(* IEC 61131-3 sources: Controller/, 6 files *)

(* ----  Codesys.ST ---- *)
(* ============================================
   КЕРУВАННЯ БОЙЛЕРОМ / ГАЗОВИМ ОБЛАДНАННЯМ
   Codesys 3.5 — Structured Text (ST)

   Як створити проект в Codesys:
   1. File → New Project → Standard Project
   2. Вибрати свій контролер або "CODESYS Control Win" для симуляції
   3. У дереві проекту: двічі клікнути PLC_PRG
   4. Вставити цей код
   5. Build → Build Solution (F11)
   6. Online → Login (Alt+F8) → Start (F5)
   ============================================ *)

PROGRAM PLC_PRG
VAR
    (* ==========================================
       АНАЛОГОВІ ВХОДИ (підключаються через
       Codesys I/O Mapping до реальних каналів)
       ========================================== *)
    AI_NAPRUGA      : INT;   (* Напруга бойлера, АЦП 0-4095 = 0-500В *)
    AI_TEMP_BOILER  : INT;   (* Температура бойлера, АЦП 0-4095 = 0-150°C *)
    AI_TEMP_VODA    : INT;   (* Температура води, АЦП 0-4095 = 0-150°C *)
    AI_TEMP_2       : INT;   (* Додатковий датчик температури *)
    AI_TISK_MASLA   : INT;   (* Тиск масла аналоговий, АЦП 0-4095 *)

    (* ==========================================
       ДИСКРЕТНІ ВХОДИ
       ========================================== *)
    X_GAZ           : BOOL;  (* Датчик газу: TRUE=є газ (замкнутий) *)
    X_VAKUUM        : BOOL;  (* Датчик вакууму: TRUE=є вакуум (замкнутий) *)
    X_TISK_MASLA_DI : BOOL;  (* Тиск масла: TRUE=норма (замкнутий) *)
    X_AVARIA_EXT    : BOOL;  (* Зовнішній аварійний СТОП *)

    (* ==========================================
       ДИСКРЕТНІ ВИХОДИ
       ========================================== *)
    Y_KLAPAN_GAZ    : BOOL;  (* Клапан газу: TRUE=відкрито *)
    Y_ROZET_1       : BOOL;  (* Розетка 1 *)
    Y_ROZET_2       : BOOL;  (* Розетка 2 *)
    Y_AVARIA_SIGNAL : BOOL;  (* Аварійна сигналізація (лампа/сирена) *)
    Y_DOZV_ROBOTY   : BOOL;  (* Загальний дозвіл роботи *)

    (* ==========================================
       КОМАНДИ ОПЕРАТОРА (з HMI або Visualization)
       ========================================== *)
    CMD_START       : BOOL;  (* Кнопка СТАРТ *)
    CMD_STOP        : BOOL;  (* Кнопка СТОП *)
    CMD_ROZET_1     : BOOL;  (* Команда увімкнути розетку 1 *)
    CMD_ROZET_2     : BOOL;  (* Команда увімкнути розетку 2 *)
    CMD_RESET_AVAR  : BOOL;  (* Скидання аварії вручну *)

    (* ==========================================
       ВНУТРІШНІ ЗМІННІ — АВАРІЇ
       ========================================== *)
    M_AVARIA_NAPRUGA    : BOOL;  (* Аварія: напруга >= 400В *)
    M_AVARIA_TEMP       : BOOL;  (* Аварія: температура бойлера >= 80°C *)
    M_AVARIA_VAKUUM     : BOOL;  (* Аварія: пропав вакуум *)
    M_ZAGALNA_AVARIA    : BOOL;  (* Загальна аварія (будь-яка з вище) *)

    (* ==========================================
       ВНУТРІШНІ ЗМІННІ — СТАНИ ДАТЧИКІВ
       ========================================== *)
    M_GAZ_IE            : BOOL;  (* Газ є = TRUE, немає = FALSE *)
    M_VAKUUM_IE         : BOOL;  (* Вакуум є = TRUE, немає = FALSE *)
    M_TISK_NORMA        : BOOL;  (* Тиск масла норма = TRUE *)

    (* ==========================================
       ВНУТРІШНІ ЗМІННІ — СИСТЕМА
       ========================================== *)
    M_SYSTEM_ON         : BOOL;  (* Система запущена оператором *)
    M_SYSTEM_READY      : BOOL;  (* Система готова до роботи *)

    (* ==========================================
       РЕАЛЬНІ ЗНАЧЕННЯ ДЛЯ ВІДОБРАЖЕННЯ НА HMI
       ========================================== *)
    NAPRUGA_VOLT        : INT;   (* Напруга в Вольтах *)
    TEMP_BOILER_GRAD    : INT;   (* Температура бойлера в °C *)
    TEMP_VODA_GRAD      : INT;   (* Температура води в °C *)
    TEMP_2_GRAD         : INT;   (* Температура доп. датчика в °C *)

    (* ==========================================
       ДОПОМІЖНІ ТРИГЕРИ (для кнопок START/STOP)
       ========================================== *)
    trig_START          : R_TRIG;  (* Фронт сигналу СТАРТ *)
    trig_STOP           : R_TRIG;  (* Фронт сигналу СТОП *)
    trig_RESET          : R_TRIG;  (* Фронт сигналу СКИДАННЯ *)
END_VAR

(* ============================================================
   БЛОК 1: ОБРОБКА КНОПОК СТАРТ / СТОП
   R_TRIG реагує тільки на момент натискання (фронт сигналу)
   ============================================================ *)
trig_START(CLK := CMD_START);
trig_STOP(CLK  := CMD_STOP);
trig_RESET(CLK := CMD_RESET_AVAR);

(* Запуск системи — тільки якщо немає аварії *)
IF trig_START.Q AND NOT M_ZAGALNA_AVARIA THEN
    M_SYSTEM_ON := TRUE;
END_IF;

(* Зупинка системи *)
IF trig_STOP.Q OR M_ZAGALNA_AVARIA THEN
    M_SYSTEM_ON := FALSE;
END_IF;

(* ============================================================
   БЛОК 2: ПЕРЕРАХУНОК АЦП → РЕАЛЬНІ ОДИНИЦІ

   Формула: РЕАЛЬНЕ = АЦП_ЗНАЧЕННЯ * МАКСИМУМ / 4095

   АЦП дає число від 0 до 4095 (12-бітний)
   Це число відповідає реальному вхідному сигналу 0-10В або 4-20мА
   ============================================================ *)

(* Напруга бойлера: вхід 0-10В = 0-500В реальних *)
NAPRUGA_VOLT     := INT_TO_INT(REAL_TO_INT(INT_TO_REAL(AI_NAPRUGA) * 500.0 / 4095.0));

(* Температура бойлера: вхід 4-20мА через модуль = 0-150°C *)
TEMP_BOILER_GRAD := INT_TO_INT(REAL_TO_INT(INT_TO_REAL(AI_TEMP_BOILER) * 150.0 / 4095.0));

(* Температура води *)
TEMP_VODA_GRAD   := INT_TO_INT(REAL_TO_INT(INT_TO_REAL(AI_TEMP_VODA) * 150.0 / 4095.0));

(* Додатковий датчик температури *)
TEMP_2_GRAD      := INT_TO_INT(REAL_TO_INT(INT_TO_REAL(AI_TEMP_2) * 150.0 / 4095.0));

(* ============================================================
   БЛОК 3: АВАРІЯ ПО НАПРУЗІ БОЙЛЕРА

   УМОВА: якщо напруга >= 400В → АВАРІЯ → все зупиняється
   ГІСТЕРЕЗИС: скидається тільки якщо впала нижче 380В
   (щоб уникнути постійного вмикання/вимикання на межі 400В)
   ============================================================ *)
IF NAPRUGA_VOLT >= 400 THEN
    M_AVARIA_NAPRUGA := TRUE;
ELSIF NAPRUGA_VOLT < 380 THEN
    (* Скидати аварію автоматично тільки якщо напруга впала *)
    (* Якщо хочеш скидати тільки вручну — закоментуй цей рядок *)
    IF trig_RESET.Q THEN
        M_AVARIA_NAPRUGA := FALSE;
    END_IF;
END_IF;

(* ============================================================
   БЛОК 4: АВАРІЯ ПО ТЕМПЕРАТУРІ БОЙЛЕРА

   УМОВА: якщо температура >= 80°C → АВАРІЯ → все зупиняється
   ГІСТЕРЕЗИС: скидається тільки якщо охолонув нижче 75°C
   ============================================================ *)
IF TEMP_BOILER_GRAD >= 80 THEN
    M_AVARIA_TEMP := TRUE;
ELSIF TEMP_BOILER_GRAD < 75 THEN
    IF trig_RESET.Q THEN
        M_AVARIA_TEMP := FALSE;
    END_IF;
END_IF;

(* ============================================================
   БЛОК 5: ДАТЧИК ГАЗУ

   X_GAZ = TRUE  (замкнутий контакт) → газ є   → M_GAZ_IE = 1
   X_GAZ = FALSE (розімкнутий)       → газу немає → M_GAZ_IE = 0

   На HMI відображати: якщо M_GAZ_IE=TRUE показуй "1 - ГАЗ Є"
                        якщо M_GAZ_IE=FALSE показуй "0 - ГАЗУ НЕМАЄ"
   ============================================================ *)
M_GAZ_IE := X_GAZ;

(* ============================================================
   БЛОК 6: ДАТЧИК ВАКУУМУ

   X_VAKUUM = TRUE  (замкнутий) → вакуум є   → робота дозволена
   X_VAKUUM = FALSE (розімкнутий) → вакууму немає → ЗУПИНКА + ЗАКРИТИ ГАЗ
   ============================================================ *)
M_VAKUUM_IE := X_VAKUUM;

IF NOT M_VAKUUM_IE THEN
    M_AVARIA_VAKUUM := TRUE;   (* Немає вакууму — АВАРІЯ *)
ELSE
    M_AVARIA_VAKUUM := FALSE;  (* Вакуум є — норма *)
END_IF;

(* ============================================================
   БЛОК 7: ДАТЧИК ТИСКУ МАСЛА

   X_TISK_MASLA_DI = TRUE  (замкнутий) → тиск норма
   X_TISK_MASLA_DI = FALSE (розімкнутий) → тиск низький → АВАРІЯ
   ============================================================ *)
M_TISK_NORMA := X_TISK_MASLA_DI;

(* ============================================================
   БЛОК 8: ЗАГАЛЬНА АВАРІЯ

   Якщо БУДЬ-ЯКА з умов виконана → загальна аварія
   → система зупиняється
   → клапан газу закривається
   → вмикається сигналізація
   ============================================================ *)
M_ZAGALNA_AVARIA := M_AVARIA_NAPRUGA    (* Напруга >= 400В *)
                 OR M_AVARIA_TEMP        (* Температура >= 80°C *)
                 OR M_AVARIA_VAKUUM      (* Немає вакууму *)
                 OR NOT M_TISK_NORMA     (* Тиск масла низький *)
                 OR X_AVARIA_EXT;        (* Зовнішній аварійний стоп *)

(* ============================================================
   БЛОК 9: ГОТОВНІСТЬ СИСТЕМИ ДО РОБОТИ

   ВСІ умови мають бути виконані одночасно:
   ✓ Напруга норма (< 400В)
   ✓ Температура норма (< 80°C)
   ✓ Газ є
   ✓ Вакуум є  ← НАЙВАЖЛИВІШЕ
   ✓ Тиск масла норма
   ✓ Немає зовнішньої аварії
   ✓ Оператор натиснув СТАРТ
   ============================================================ *)
M_SYSTEM_READY := NOT M_AVARIA_NAPRUGA
              AND NOT M_AVARIA_TEMP
              AND M_GAZ_IE
              AND M_VAKUUM_IE
              AND M_TISK_NORMA
              AND NOT X_AVARIA_EXT
              AND M_SYSTEM_ON;

(* ============================================================
   БЛОК 10: КЕРУВАННЯ КЛАПАНОМ ГАЗУ

   ВІДКРИТИ газ → тільки якщо система готова (всі умови ОК)
   ЗАКРИТИ газ → при будь-якій аварії, і особливо при відсутності вакууму

   БЕЗПЕКА: подвійна перевірка вакууму — навіть якщо
   щось пішло не так в логіці вище, газ все одно закриється
   ============================================================ *)
IF M_SYSTEM_READY THEN
    Y_KLAPAN_GAZ := TRUE;    (* Відкрити клапан газу *)
ELSE
    Y_KLAPAN_GAZ := FALSE;   (* Закрити клапан газу *)
END_IF;

(* КРИТИЧНА БЕЗПЕКА: подвійна гарантія закриття газу без вакууму *)
IF NOT M_VAKUUM_IE THEN
    Y_KLAPAN_GAZ := FALSE;   (* ОБОВ'ЯЗКОВО закрити! *)
END_IF;

(* КРИТИЧНА БЕЗПЕКА: закрити газ при аварії напруги або температури *)
IF M_AVARIA_NAPRUGA OR M_AVARIA_TEMP THEN
    Y_KLAPAN_GAZ := FALSE;
END_IF;

(* ============================================================
   БЛОК 11: КЕРУВАННЯ РОЗЕТКАМИ

   Розетки вмикаються командою оператора (з HMI або кнопки)
   АЛЕ тільки якщо немає загальної аварії
   ============================================================ *)
IF CMD_ROZET_1 AND NOT M_ZAGALNA_AVARIA THEN
    Y_ROZET_1 := TRUE;
ELSE
    Y_ROZET_1 := FALSE;
END_IF;

IF CMD_ROZET_2 AND NOT M_ZAGALNA_AVARIA THEN
    Y_ROZET_2 := TRUE;
ELSE
    Y_ROZET_2 := FALSE;
END_IF;

(* ============================================================
   БЛОК 12: АВАРІЙНА СИГНАЛІЗАЦІЯ
   Лампа або сирена вмикається при будь-якій аварії
   ============================================================ *)
Y_AVARIA_SIGNAL := M_ZAGALNA_AVARIA;

(* ============================================================
   БЛОК 13: ЗАГАЛЬНИЙ ДОЗВІЛ РОБОТИ
   Цей вихід можна підключити до загального контактора
   ============================================================ *)
Y_DOZV_ROBOTY := M_SYSTEM_READY;

END_PROGRAM

(* ---- BoilerController.ST ---- *)
(* ============================================
   КОНТРОЛЕР УПРАВЛІННЯ БОЙЛЕРОМ
   FATEK FBs-MA - Structured Text (ST)
   Версія 2.0 - Оптимізований під ваші вимоги
   ============================================ *)

(* --- КОНСТАНТИ --- *)
VAR CONSTANT
    (* Діапазони АЦП *)
    ADC_MAX         : INT := 4095;
    VOLTAGE_MAX     : INT := 500;   (* Макс. напруга, В *)
    TEMP_MAX        : INT := 150;   (* Макс. температура, °C *)

    (* Аварійні межі *)
    VOLTAGE_ALARM   : INT := 400;   (* Аварія напруги при 400В *)
    VOLTAGE_RESET   : INT := 380;   (* Скидання при 380В *)
    TEMP_ALARM      : INT := 80;    (* Аварія температури при 80°C *)
    TEMP_RESET      : INT := 75;    (* Скидання при 75°C *)

    (* АЦП значення для аварій *)
    ADC_VOLTAGE_ALARM : INT := 3276; (* 400В → АЦП: 4095*400/500 *)
    ADC_TEMP_ALARM    : INT := 2184; (* 80°C → АЦП: 4095*80/150 *)
END_VAR

(* --- ВХОДИ (Inputs) --- *)
VAR
    (* Аналогові входи 0..4095 *)
    AI_VOLTAGE      AT %IW0 : INT;   (* Напруга бойлера 0-500В *)
    AI_TEMP_BOILER  AT %IW1 : INT;   (* Температура бойлера 0-150°C *)
    AI_TEMP_WATER   AT %IW2 : INT;   (* Температура води 0-150°C *)
    AI_TEMP_1       AT %IW3 : INT;   (* Датчик температури 1 *)
    AI_TEMP_2       AT %IW4 : INT;   (* Датчик температури 2 *)
    AI_OIL_PRESSURE AT %IW5 : INT;   (* Тиск масла (аналоговий) *)

    (* Дискретні входи *)
    X_GAS_PRESENT   AT %IX0.0 : BOOL; (* Датчик газу: TRUE=є газ *)
    X_VACUUM_OK     AT %IX0.1 : BOOL; (* Датчик вакууму: TRUE=є вакуум *)
    X_OIL_PRESS_OK  AT %IX0.2 : BOOL; (* Тиск масла: TRUE=норма *)
    X_EMERGENCY_STOP: AT %IX0.3 : BOOL; (* Аварійний стоп: TRUE=активний *)

    (* Команди оператора/HMI *)
    CMD_START       AT %MX10.0 : BOOL; (* Команда старт *)
    CMD_STOP        AT %MX10.1 : BOOL; (* Команда стоп *)
    CMD_SOCKET1     AT %MX10.2 : BOOL; (* Команда розетка 1 *)
    CMD_SOCKET2     AT %MX10.3 : BOOL; (* Команда розетка 2 *)
END_VAR

(* --- ВИХОДИ (Outputs) --- *)
VAR
    Y_GAS_VALVE     AT %QX0.0 : BOOL; (* Клапан газу: TRUE=відкрито *)
    Y_SOCKET1       AT %QX0.1 : BOOL; (* Розетка 1 *)
    Y_SOCKET2       AT %QX0.2 : BOOL; (* Розетка 2 *)
    Y_ALARM_LIGHT   AT %QX0.3 : BOOL; (* Аварійна лампа *)
    Y_PERMIT_RUN    AT %QX0.4 : BOOL; (* Дозвіл роботи *)
    Y_WATER_PUMP    AT %QX0.5 : BOOL; (* Насос води *)
END_VAR

(* --- ВНУТРІШНІ МАРКЕРИ --- *)
VAR
    (* Аварійні флаги *)
    M_VOLTAGE_ALARM : BOOL := FALSE; (* Аварія напруги *)
    M_TEMP_ALARM    : BOOL := FALSE; (* Аварія температури *)
    M_VACUUM_ALARM  : BOOL := FALSE; (* Аварія вакууму *)
    M_OIL_ALARM     : BOOL := FALSE; (* Аварія тиску масла *)
    M_ANY_ALARM     : BOOL := FALSE; (* Будь-яка аварія *)

    (* Стан системи *)
    M_SYSTEM_RUN    : BOOL := FALSE; (* Система запущена *)
    M_SYSTEM_READY  : BOOL := FALSE; (* Система готова *)
    M_GAS_AVAILABLE : BOOL := FALSE; (* Газ доступний *)
    M_VACUUM_OK     : BOOL := FALSE; (* Вакуум в нормі *)

    (* Фізичні величини для HMI *)
    VOLTAGE_DISPLAY : INT; (* Напруга в Вольтах *)
    TEMP_B_DISPLAY  : INT; (* Температура бойлера °C *)
    TEMP_W_DISPLAY  : INT; (* Температура води °C *)
    TEMP_1_DISPLAY  : INT; (* Температура датчик 1 °C *)
    TEMP_2_DISPLAY  : INT; (* Температура датчик 2 °C *)
    OIL_P_DISPLAY   : INT; (* Тиск масла в ум.од.*)

    (* Детектори фронтів *)
    M_CMD_START_OLD : BOOL := FALSE;
    M_CMD_STOP_OLD  : BOOL := FALSE;
    M_GAS_OLD       : BOOL := FALSE;
    M_VAC_OLD       : BOOL := FALSE;
    M_ALARM_OLD     : BOOL := FALSE;

    (* Статистика для HMI *)
    STAT_START_COUNT: INT := 0;
    STAT_ALARM_COUNT: INT := 0;
    STAT_GAS_OFF    : INT := 0;
    STAT_VAC_OFF    : INT := 0;
END_VAR

(* ============================================
   БЛОК 1: ПЕРЕТВОРЕННЯ АЦП → ФІЗИЧНІ ВЕЛИЧИНИ
   ============================================ *)

(* Напруга: 0-4095 = 0-500В *)
VOLTAGE_DISPLAY := AI_VOLTAGE * VOLTAGE_MAX / ADC_MAX;

(* Температури: 0-4095 = 0-150°C *)
TEMP_B_DISPLAY := AI_TEMP_BOILER * TEMP_MAX / ADC_MAX;
TEMP_W_DISPLAY := AI_TEMP_WATER * TEMP_MAX / ADC_MAX;
TEMP_1_DISPLAY := AI_TEMP_1 * TEMP_MAX / ADC_MAX;
TEMP_2_DISPLAY := AI_TEMP_2 * TEMP_MAX / ADC_MAX;

(* Тиск масла: 0-4095 = 0-100% *)
OIL_P_DISPLAY := AI_OIL_PRESSURE * 100 / ADC_MAX;

(* ============================================
   БЛОК 2: АВАРІЯ НАПРУГИ (≥400В)
   ============================================ *)
IF VOLTAGE_DISPLAY >= VOLTAGE_ALARM THEN
    M_VOLTAGE_ALARM := TRUE;
ELSE
    IF VOLTAGE_DISPLAY < VOLTAGE_RESET THEN
        M_VOLTAGE_ALARM := FALSE;
    END_IF;
END_IF;

(* ============================================
   БЛОК 3: АВАРІЯ ТЕМПЕРАТУРИ (≥80°C)
   ============================================ *)
IF TEMP_B_DISPLAY >= TEMP_ALARM THEN
    M_TEMP_ALARM := TRUE;
ELSE
    IF TEMP_B_DISPLAY < TEMP_RESET THEN
        M_TEMP_ALARM := FALSE;
    END_IF;
END_IF;

(* ============================================
   БЛОК 4: ДАТЧИК ГАЗУ
   ============================================ *)
M_GAS_AVAILABLE := X_GAS_PRESENT;

(* Лічильник відключень газу *)
IF M_GAS_AVAILABLE = FALSE AND M_GAS_OLD = TRUE THEN
    STAT_GAS_OFF := STAT_GAS_OFF + 1;
END_IF;
M_GAS_OLD := M_GAS_AVAILABLE;

(* ============================================
   БЛОК 5: ДАТЧИК ВАКУУМУ
   ============================================ *)
M_VACUUM_OK := X_VACUUM_OK;

IF M_VACUUM_OK = FALSE THEN
    M_VACUUM_ALARM := TRUE;  (* Немає вакууму = аварія *)
ELSE
    M_VACUUM_ALARM := FALSE;
END_IF;

(* Лічильник відключень вакууму *)
IF M_VACUUM_OK = FALSE AND M_VAC_OLD = TRUE THEN
    STAT_VAC_OFF := STAT_VAC_OFF + 1;
END_IF;
M_VAC_OLD := M_VACUUM_OK;

(* ============================================
   БЛОК 6: ТИСК МАСЛА
   ============================================ *)
IF X_OIL_PRESS_OK = FALSE THEN
    M_OIL_ALARM := TRUE;
ELSE
    M_OIL_ALARM := FALSE;
END_IF;

(* ============================================
   БЛОК 7: ЗАГАЛЬНА АВАРІЯ
   ============================================ *)
M_ANY_ALARM := M_VOLTAGE_ALARM
             OR M_TEMP_ALARM
             OR M_VACUUM_ALARM
             OR M_OIL_ALARM
             OR X_EMERGENCY_STOP;

(* Лічильник аварій *)
IF M_ANY_ALARM = TRUE AND M_ALARM_OLD = FALSE THEN
    STAT_ALARM_COUNT := STAT_ALARM_COUNT + 1;
END_IF;
M_ALARM_OLD := M_ANY_ALARM;

(* ============================================
   БЛОК 8: ЛОГІКА СТАРТ/СТОП
   ============================================ *)

(* Детектор фронту старту *)
IF CMD_START = TRUE AND M_CMD_START_OLD = FALSE THEN
    IF M_SYSTEM_RUN = FALSE AND M_ANY_ALARM = FALSE THEN
        M_SYSTEM_RUN := TRUE;
        STAT_START_COUNT := STAT_START_COUNT + 1;
    END_IF;
END_IF;
M_CMD_START_OLD := CMD_START;

(* Детектор фронту стопу *)
IF CMD_STOP = TRUE AND M_CMD_STOP_OLD = FALSE THEN
    M_SYSTEM_RUN := FALSE;
END_IF;
M_CMD_STOP_OLD := CMD_STOP;

(* Автоматичний стоп при аварії *)
IF M_ANY_ALARM = TRUE THEN
    M_SYSTEM_RUN := FALSE;
END_IF;

(* ============================================
   БЛОК 9: ГОТОВНІСТЬ СИСТЕМИ
   ============================================ *)
M_SYSTEM_READY := NOT M_VOLTAGE_ALARM      (* Напруга норма *)
                AND NOT M_TEMP_ALARM        (* Температура норма *)
                AND M_GAS_AVAILABLE          (* Газ є *)
                AND M_VACUUM_OK              (* Вакуум є *)
                AND NOT M_OIL_ALARM           (* Тиск масла норма *)
                AND NOT X_EMERGENCY_STOP      (* Немає аварійного стопу *)
                AND M_SYSTEM_RUN;             (* Система запущена *)

(* ============================================
   БЛОК 10: КЕРУВАННЯ КЛАПАНОМ ГАЗУ
   ============================================ *)
(* Головна логіка: газ відкритий тільки якщо ВСІ умови виконані *)
IF M_SYSTEM_READY THEN
    Y_GAS_VALVE := TRUE;   (* Відкрити клапан газу *)
ELSE
    Y_GAS_VALVE := FALSE;  (* Закрити клапан газу *)
END_IF;

(* Додатковий захист: якщо немає вакууму - ОБОВ'ЯЗКОВО закрити газ *)
IF M_VACUUM_OK = FALSE THEN
    Y_GAS_VALVE := FALSE;
END_IF;

(* ============================================
   БЛОК 11: КЕРУВАННЯ РОЗЕТКАМИ
   ============================================ *)

(* Розетка 1 - вмикається командою, але не при аварії *)
IF CMD_SOCKET1 = TRUE AND M_ANY_ALARM = FALSE THEN
    Y_SOCKET1 := TRUE;
ELSE
    Y_SOCKET1 := FALSE;
END_IF;

(* Розетка 2 - вмикається командою, але не при аварії *)
IF CMD_SOCKET2 = TRUE AND M_ANY_ALARM = FALSE THEN
    Y_SOCKET2 := TRUE;
ELSE
    Y_SOCKET2 := FALSE;
END_IF;

(* ============================================
   БЛОК 12: КЕРУВАННЯ НАСОСОМ ВОДИ
   ============================================ *)
(* Насос води працює якщо система готова і є температура води *)
IF M_SYSTEM_READY AND TEMP_W_DISPLAY > 20 THEN
    Y_WATER_PUMP := TRUE;
ELSE
    Y_WATER_PUMP := FALSE;
END_IF;

(* ============================================
   БЛОК 13: АВАРІЙНА СИГНАЛІЗАЦІЯ
   ============================================ *)
Y_ALARM_LIGHT := M_ANY_ALARM;

(* ============================================
   БЛОК 14: ЗАГАЛЬНИЙ ДОЗВІЛ РОБОТИ
   ============================================ *)
Y_PERMIT_RUN := M_SYSTEM_READY;

(* ============================================
   БЛОК 15: ЕКСПОРТ ДАНИХ ДЛЯ HMI
   ============================================ *)
(* Ці маркери можна використовувати для відображення на HMI дисплей *)
(*
MW0  = VOLTAGE_DISPLAY    (* Напруга в Вольтах *)
MW1  = TEMP_B_DISPLAY     (* Температура бойлера °C *)
MW2  = TEMP_W_DISPLAY     (* Температура води °C *)
MW3  = TEMP_1_DISPLAY     (* Температура датчик 1 °C *)
MW4  = TEMP_2_DISPLAY     (* Температура датчик 2 °C *)
MW5  = OIL_P_DISPLAY      (* Тиск масла % *)

MW10 = STAT_START_COUNT   (* Кількість запусків *)
MW11 = STAT_ALARM_COUNT   (* Кількість аварій *)
MW12 = STAT_GAS_OFF       (* Відключень газу *)
MW13 = STAT_VAC_OFF       (* Відключень вакууму *)

MX20 = M_SYSTEM_RUN       (* Система запущена *)
MX21 = M_SYSTEM_READY     (* Система готова *)
MX22 = M_GAS_AVAILABLE    (* Газ доступний *)
MX23 = M_VACUUM_OK        (* Вакуум в нормі *)
MX24 = M_VOLTAGE_ALARM    (* Аварія напруги *)
MX25 = M_TEMP_ALARM       (* Аварія температури *)
MX26 = M_VACUUM_ALARM     (* Аварія вакууму *)
MX27 = M_OIL_ALARM        (* Аварія тиску масла *)
MX28 = M_ANY_ALARM        (* Загальна аварія *)
*)

(* ---- Controller.ST ---- *)
(* ============================================
   КЕРУВАННЯ БОЙЛЕРОМ / ГАЗОВИМ ОБЛАДНАННЯМ
   Fatek FBs-MA — Structured Text (ST)
   Повна версія з усіма функціями з Python-коду
   ============================================ *)

(* --- КОНСТАНТИ --- *)
VAR CONSTANT
    (* Межі АЦП *)
    ADC_MAX             : INT := 4095;
    NAPRUGA_MAX         : INT := 500;   (* Макс. напруга, В *)
    TEMP_MAX            : INT := 150;   (* Макс. температура, °C *)

    (* Межі спрацьовування аварій *)
    NAPRUGA_AVAR_VOLT   : INT := 400;   (* Аварія напруги при 400В *)
    NAPRUGA_HYST_VOLT   : INT := 380;   (* Гістерезис: скидання при 380В *)
    TEMP_AVAR_GRAD      : INT := 80;    (* Аварія температури при 80°C *)
    TEMP_HYST_GRAD      : INT := 75;    (* Гістерезис: скидання при 75°C *)

    (* Відповідні значення АЦП для аварій *)
    NAPRUGA_AVARIA      : INT := 3276;  (* 400В → АЦП: 4095*400/500=3276 *)
    TEMP_BOILER_AVARIA  : INT := 2184;  (* 80°C → АЦП: 4095*80/150=2184 *)
END_VAR

(* --- ЗМІННІ ВХОДІВ (Inputs) --- *)
VAR
    (* Аналогові входи 0..4095 *)
    AI_NAPRUGA      AT %IW0 : INT;   (* Напруга бойлера 0-500В *)
    AI_TEMP_BOILER  AT %IW1 : INT;   (* Температура бойлера 0-150°C *)
    AI_TEMP_VODA    AT %IW2 : INT;   (* Температура води 0-150°C *)
    AI_TEMP_2       AT %IW3 : INT;   (* Додатковий датчик температури *)
    AI_TISK_MASLA   AT %IW4 : INT;   (* Тиск масла (аналоговий датчик) *)

    (* Дискретні входи *)
    X_GAZ           AT %IX0.0 : BOOL; (* Датчик газу: TRUE=є газ *)
    X_VAKUUM        AT %IX0.1 : BOOL; (* Датчик вакууму: TRUE=є вакуум *)
    X_TISK_MASLA_DI AT %IX0.2 : BOOL; (* Тиск масла дискретний: TRUE=норма *)
    X_AVARIA_EXT    AT %IX0.3 : BOOL; (* Зовнішній аварійний стоп *)

    (* Команди з HMI / оператора *)
    CMD_ROZET_1     AT %MX10.0 : BOOL; (* Команда вкл. розетки 1 *)
    CMD_ROZET_2     AT %MX10.1 : BOOL; (* Команда вкл. розетки 2 *)
    CMD_START       AT %MX10.2 : BOOL; (* Старт системи (імпульс) *)
    CMD_STOP        AT %MX10.3 : BOOL; (* Стоп системи (імпульс) *)
END_VAR

(* --- ЗМІННІ ВИХОДІВ (Outputs) --- *)
VAR
    Y_KLAPAN_GAZ    AT %QX0.0 : BOOL; (* Клапан газу: TRUE=відкрито *)
    Y_ROZET_1       AT %QX0.1 : BOOL; (* Розетка 1 *)
    Y_ROZET_2       AT %QX0.2 : BOOL; (* Розетка 2 *)
    Y_AVARIA_SIGNAL AT %QX0.3 : BOOL; (* Аварійна сигналізація *)
    Y_DOZV_ROBOTY   AT %QX0.4 : BOOL; (* Загальний дозвіл роботи *)
END_VAR

(* --- ВНУТРІШНІ МАРКЕРИ --- *)
VAR
    (* Аварії *)
    M_AVARIA_NAPRUGA    : BOOL; (* Аварія: напруга >= 400В *)
    M_AVARIA_TEMP       : BOOL; (* Аварія: температура >= 80°C *)
    M_AVARIA_VAKUUM     : BOOL; (* Аварія: пропав вакуум *)
    M_ZAGALNA_AVARIA    : BOOL; (* Будь-яка аварія *)

    (* Стан датчиків *)
    M_GAZ_IE            : BOOL; (* Газ є = 1, немає = 0 *)
    M_VAKUUM_IE         : BOOL; (* Вакуум є = 1, немає = 0 *)
    M_TISK_NORMA        : BOOL; (* Тиск масла в нормі *)

    (* Стан системи *)
    M_SYSTEM_ON         : BOOL; (* Система запущена *)
    M_SYSTEM_READY      : BOOL; (* Система готова до роботи *)

    (* Фізичні величини (для відображення на HMI) *)
    TEMP_BOILER_GRAD    : INT;  (* Температура бойлера °C *)
    TEMP_VODA_GRAD      : INT;  (* Температура води °C *)
    TEMP_2_GRAD         : INT;  (* Температура доп. датчик °C *)
    NAPRUGA_VOLT        : INT;  (* Напруга в Вольтах *)

    (* Допоміжні змінні для статистики *)
    M_START_PULSE       : BOOL; (* Детектор імпульсу старту *)
    M_STOP_PULSE        : BOOL; (* Детектор імпульсу стопу *)
    STAT_STARTS         : INT;  (* Лічильник запусків *)
    STAT_STOPS          : INT;  (* Лічильник зупинок *)
    STAT_ALARMS         : INT;  (* Лічильник аварій *)
    STAT_GAS_OFF        : INT;  (* Лічильник відключень газу *)
    STAT_VAKUUM_OFF     : INT;  (* Лічильник відключень вакууму *)

    (* Для детектора фронтів *)
    M_CMD_START_OLD     : BOOL;
    M_CMD_STOP_OLD      : BOOL;
    M_GAZ_OLD           : BOOL;
    M_VAKUUM_OLD        : BOOL;
    M_ALARM_OLD         : BOOL;
END_VAR

(* ============================================
   БЛОК 1: ПЕРЕРАХУНОК АЦП → РЕАЛЬНІ ОДИНИЦІ
   Формула: РЕАЛ = АЦП * MAX_ЗНАЧЕННЯ / 4095
   ============================================ *)

(* Напруга: 0-4095 = 0-500В *)
NAPRUGA_VOLT    := AI_NAPRUGA * 500 / 4095;

(* Температури: 0-4095 = 0-150°C *)
TEMP_BOILER_GRAD := AI_TEMP_BOILER * 150 / 4095;
TEMP_VODA_GRAD   := AI_TEMP_VODA * 150 / 4095;
TEMP_2_GRAD      := AI_TEMP_2 * 150 / 4095;

(* ============================================
   БЛОК 2: АВАРІЯ ПО НАПРУЗІ БОЙЛЕРА
   З гістерезисом: ввімкнення при 400В, вимкнення при 380В
   ============================================ *)
IF NAPRUGA_VOLT >= NAPRUGA_AVAR_VOLT THEN
    M_AVARIA_NAPRUGA := TRUE;
ELSE
    IF NAPRUGA_VOLT < NAPRUGA_HYST_VOLT THEN
        M_AVARIA_NAPRUGA := FALSE;
    END_IF;
END_IF;

(* ============================================
   БЛОК 3: АВАРІЯ ПО ТЕМПЕРАТУРІ БОЙЛЕРА
   З гістерезисом: ввімкнення при 80°C, вимкнення при 75°C
   ============================================ *)
IF TEMP_BOILER_GRAD >= TEMP_AVAR_GRAD THEN
    M_AVARIA_TEMP := TRUE;
ELSE
    IF TEMP_BOILER_GRAD < TEMP_HYST_GRAD THEN
        M_AVARIA_TEMP := FALSE;
    END_IF;
END_IF;

(* ============================================
   БЛОК 4: ДАТЧИК ГАЗУ
   X_GAZ = TRUE (замкнутий) → газ є (M_GAZ_IE = 1)
   X_GAZ = FALSE (розімкнутий) → газу немає (M_GAZ_IE = 0)
   ============================================ *)
M_GAZ_IE := X_GAZ;

(* Лічильник відключень газу *)
IF M_GAZ_IE = FALSE AND M_GAZ_OLD = TRUE THEN
    STAT_GAS_OFF := STAT_GAS_OFF + 1;
END_IF;
M_GAZ_OLD := M_GAZ_IE;

(* ============================================
   БЛОК 5: ДАТЧИК ВАКУУМУ
   X_VAKUUM = TRUE (замкнутий) → вакуум є
   X_VAKUUM = FALSE (розімкнутий) → вакууму немає → АВАРІЯ
   ============================================ *)
M_VAKUUM_IE := X_VAKUUM;

IF NOT M_VAKUUM_IE THEN
    M_AVARIA_VAKUUM := TRUE;  (* Пропав вакуум — аварія *)
ELSE
    M_AVARIA_VAKUUM := FALSE; (* Вакуум є — норма *)
END_IF;

(* Лічильник відключень вакууму *)
IF M_VAKUUM_IE = FALSE AND M_VAKUUM_OLD = TRUE THEN
    STAT_VAKUUM_OFF := STAT_VAKUUM_OFF + 1;
END_IF;
M_VAKUUM_OLD := M_VAKUUM_IE;

(* ============================================
   БЛОК 6: ТИСК МАСЛА
   X_TISK_MASLA_DI = TRUE → тиск норма
   ============================================ *)
M_TISK_NORMA := X_TISK_MASLA_DI;

(* ============================================
   БЛОК 7: ЗАГАЛЬНА АВАРІЯ
   Будь-яка з умов → загальна аварія
   ============================================ *)
M_ZAGALNA_AVARIA := M_AVARIA_NAPRUGA
                 OR M_AVARIA_TEMP
                 OR M_AVARIA_VAKUUM
                 OR NOT M_TISK_NORMA
                 OR X_AVARIA_EXT;

(* Лічильник аварій (по передньому фронту) *)
IF M_ZAGALNA_AVARIA = TRUE AND M_ALARM_OLD = FALSE THEN
    STAT_ALARMS := STAT_ALARMS + 1;
END_IF;
M_ALARM_OLD := M_ZAGALNA_AVARIA;

(* ============================================
   БЛОК 8: ЛОГІКА СТАРТ/СТОП
   Детектори імпульсів та керування станом системи
   ============================================ *)

(* Детектор переднього фронту для СТАРТ *)
M_START_PULSE := CMD_START AND NOT M_CMD_START_OLD;
M_CMD_START_OLD := CMD_START;

(* Детектор переднього фронту для СТОП *)
M_STOP_PULSE := CMD_STOP AND NOT M_CMD_STOP_OLD;
M_CMD_STOP_OLD := CMD_STOP;

(* Старт системи *)
IF M_START_PULSE AND NOT M_SYSTEM_ON AND NOT M_ZAGALNA_AVARIA THEN
    M_SYSTEM_ON := TRUE;
    STAT_STARTS := STAT_STARTS + 1;
END_IF;

(* Стоп системи *)
IF M_STOP_PULSE OR M_ZAGALNA_AVARIA THEN
    IF M_SYSTEM_ON THEN
        M_SYSTEM_ON := FALSE;
        STAT_STOPS := STAT_STOPS + 1;
    END_IF;
END_IF;

(* ============================================
   БЛОК 9: ГОТОВНІСТЬ СИСТЕМИ ДО РОБОТИ
   Всі умови мають бути виконані
   ============================================ *)
M_SYSTEM_READY := NOT M_AVARIA_NAPRUGA   (* Напруга норма *)
              AND NOT M_AVARIA_TEMP       (* Температура норма *)
              AND M_GAZ_IE                (* Газ є *)
              AND M_VAKUUM_IE             (* Вакуум є *)
              AND M_TISK_NORMA            (* Тиск масла норма *)
              AND NOT X_AVARIA_EXT        (* Немає зовнішньої аварії *)
              AND M_SYSTEM_ON;            (* Система запущена *)

(* ============================================
   БЛОК 10: КЕРУВАННЯ КЛАПАНОМ ГАЗУ (Y0)
   Відкрити тільки якщо ВСІ умови виконані
   Додаткова гарантія: без вакууму газ закрито
   ============================================ *)
IF M_SYSTEM_READY THEN
    Y_KLAPAN_GAZ := TRUE;   (* Відкрити клапан газу *)
ELSE
    Y_KLAPAN_GAZ := FALSE;  (* ЗАЧИНИТИ клапан газу *)
END_IF;

(* Додаткова гарантія: якщо немає вакууму — ОБОВ'ЯЗКОВО закрити газ *)
IF NOT M_VAKUUM_IE THEN
    Y_KLAPAN_GAZ := FALSE;
END_IF;

(* ============================================
   БЛОК 11: КЕРУВАННЯ РОЗЕТКАМИ
   Вмикаються командою з контролера/HMI
   але тільки якщо немає загальної аварії
   ============================================ *)

(* Розетка 1 *)
IF CMD_ROZET_1 AND NOT M_ZAGALNA_AVARIA THEN
    Y_ROZET_1 := TRUE;
ELSE
    Y_ROZET_1 := FALSE;
END_IF;

(* Розетка 2 *)
IF CMD_ROZET_2 AND NOT M_ZAGALNA_AVARIA THEN
    Y_ROZET_2 := TRUE;
ELSE
    Y_ROZET_2 := FALSE;
END_IF;

(* ============================================
   БЛОК 12: АВАРІЙНА СИГНАЛІЗАЦІЯ
   ============================================ *)
Y_AVARIA_SIGNAL := M_ZAGALNA_AVARIA;

(* ============================================
   БЛОК 13: ЗАГАЛЬНИЙ ДОЗВІЛ РОБОТИ
   ============================================ *)
Y_DOZV_ROBOTY := M_SYSTEM_READY;

(* ============================================
   БЛОК 14: СТАТИСТИКА ДЛЯ HMI
   Виведення на HMI дисплей
   ============================================ *)

(* Маркери для відображення на HMI *)
(*
   MW0  = NAPRUGA_VOLT      (відображати в Вольтах)
   MW1  = TEMP_BOILER_GRAD  (відображати в °C)
   MW2  = TEMP_VODA_GRAD    (відображати в °C)
   MW3  = TEMP_2_GRAD       (відображати в °C)
   MW10 = STAT_STARTS       (кількість запусків)
   MW11 = STAT_STOPS        (кількість зупинок)
   MW12 = STAT_ALARMS       (кількість аварій)
   MW13 = STAT_GAS_OFF      (скільки разів відключався газ)
   MW14 = STAT_VAKUUM_OFF   (скільки разів пропадав вакуум)
*)

(* ---- FATEK_BoilerControl.ST ---- *)
(* ============================================
   ПРОГРАМА КОНТРОЛЕРА БОЙЛЕРА
   Для FATEK FBs-10MAR
   Structured Text (ST) - готовий до завантаження
   ============================================ *)

PROGRAM BoilerControl

(* --- КОНСТАНТИ СИСТЕМИ --- *)
VAR_CONSTANT
    ADC_MAX         : INT := 4095;          (* Максимальне значення АЦП *)
    VOLTAGE_MAX     : INT := 500;           (* Макс. напруга 500В *)
    TEMP_MAX        : INT := 150;           (* Макс. температура 150°C *)

    (* Аварійні пороги *)
    VOLTAGE_TRIP    : INT := 400;           (* Відключення при 400В *)
    VOLTAGE_RESET   : INT := 380;           (* Відновлення при 380В *)
    TEMP_TRIP       : INT := 80;            (* Відключення при 80°C *)
    TEMP_RESET      : INT := 75;            (* Відновлення при 75°C *)
END_VAR

(* --- ВХОДИ (INPUTS) --- *)
VAR
    (* Аналогові входи FBs-10MAR *)
    AI_BoilerVoltage    AT %IW0 : INT;      (* Напруга бойлера 0-500В *)
    AI_BoilerTemp       AT %IW1 : INT;      (* Температура бойлера 0-150°C *)
    AI_WaterTemp        AT %IW2 : INT;      (* Температура води 0-150°C *)
    AI_TempSensor1      AT %IW3 : INT;      (* Датчик температури 1 *)
    AI_TempSensor2      AT %IW4 : INT;      (* Датчик температури 2 *)
    AI_OilPressure      AT %IW5 : INT;      (* Тиск масла 0-100% *)
    AI_SteamPressure    AT %IW6 : INT;      (* Тиск пари 0-10 бар *)

    (* Дискретні входи *)
    DI_GasSensor        AT %IX0.0 : BOOL;    (* Датчик газу: 1=є, 0=немає *)
    DI_VacuumSensor     AT %IX0.1 : BOOL;    (* Датчик вакууму: 1=є, 0=немає *)
    DI_OilPressureOK    AT %IX0.2 : BOOL;    (* Тиск масла: 1=норма, 0=низький *)
    DI_SteamPressureOK  AT %IX0.3 : BOOL;    (* Тиск пари: 1=норма, 0=високий/низький *)
    DI_EmergencyStop    AT %IX0.4 : BOOL;    (* Аварійний стоп: 1=активний *)
    DI_ManualMode       AT %IX0.5 : BOOL;    (* Ручний режим: 1=вкл *)

    (* Команди з панелі оператора *)
    CMD_SystemStart      AT %MX0.0 : BOOL;    (* Старт системи *)
    CMD_SystemStop       AT %MX0.1 : BOOL;    (* Стоп системи *)
    CMD_Socket1_On       AT %MX0.2 : BOOL;    (* Вкл розетку 1 *)
    CMD_Socket2_On       AT %MX0.3 : BOOL;    (* Вкл розетку 2 *)
    CMD_ResetAlarms      AT %MX0.4 : BOOL;    (* Скидання аварій *)
END_VAR

(* --- ВИХОДИ (OUTPUTS) --- *)
VAR
    (* Керуючі виходи *)
    DO_GasValve         AT %QX0.0 : BOOL;    (* Клапан газу: 1=відкрито *)
    DO_Socket1          AT %QX0.1 : BOOL;    (* Розетка 1: 1=вкл *)
    DO_Socket2          AT %QX0.2 : BOOL;    (* Розетка 2: 1=вкл *)
    DO_WaterPump        AT %QX0.3 : BOOL;    (* Насос води: 1=вкл *)
    DO_OilPump          AT %QX0.4 : BOOL;    (* Насос масла: 1=вкл *)
    DO_AlarmLight       AT %QX0.5 : BOOL;    (* Аварійна лампа: 1=вкл *)
    DO_PermitRun        AT %QX0.6 : BOOL;    (* Дозвіл роботи: 1=дозволено *)
    DO_FanVent          AT %QX0.7 : BOOL;    (* Вентиляція: 1=вкл *)

    (* Індикація стану для HMI *)
    ST_SystemRunning    AT %QW0 : INT;       (* Стан системи *)
    ST_GasAvailable     AT %QW1 : INT;       (* Наявність газу: 1/0 *)
    ST_VacuumOK         AT %QW2 : INT;       (* Вакуум: 1/0 *)
    ST_AlarmCode        AT %QW3 : INT;       (* Код аварії *)
END_VAR

(* --- ВНУТРІШНІ МАРКЕРИ --- *)
VAR
    (* Аварійні флаги *)
    ALM_VoltageHigh     : BOOL := FALSE;     (* Аварія: висока напруга *)
    ALM_TempHigh        : BOOL := FALSE;     (* Аварія: висока температура *)
    ALM_NoGas           : BOOL := FALSE;     (* Аварія: немає газу *)
    ALM_NoVacuum        : BOOL := FALSE;     (* Аварія: немає вакууму *)
    ALM_OilPressureLow  : BOOL := FALSE;     (* Аварія: низький тиск масла *)
    ALM_SteamPressureBad: BOOL := FALSE;     (* Аварія: неправильний тиск пари *)
    ALM_Emergency       : BOOL := FALSE;     (* Аварія: аварійний стоп *)
    ALM_AnyAlarm        : BOOL := FALSE;     (* Будь-яка аварія *)

    (* Стан системи *)
    SYS_Enabled         : BOOL := FALSE;     (* Система дозволена *)
    SYS_Running         : BOOL := FALSE;     (* Система працює *)
    SYS_Ready           : BOOL := FALSE;     (* Система готова *)
    SYS_ManualMode      : BOOL := FALSE;     (* Ручний режим *)

    (* Стан датчиків *)
    SNS_GasPresent      : BOOL := FALSE;     (* Газ присутній *)
    SNS_VacuumPresent   : BOOL := FALSE;     (* Вакуум присутній *)
    SNS_OilPressureOK   : BOOL := FALSE;     (* Тиск масла норма *)
    SNS_SteamPressureOK : BOOL := FALSE;     (* Тиск пари норма *)

    (* Фізичні величини для відображення *)
    PHY_Voltage         : INT;               (* Напруга в Вольтах *)
    PHY_BoilerTemp      : INT;               (* Температура бойлера °C *)
    PHY_WaterTemp       : INT;               (* Температура води °C *)
    PHY_Temp1           : INT;               (* Температура датчик 1 °C *)
    PHY_Temp2           : INT;               (* Температура датчик 2 °C *)
    PHY_OilPressure     : INT;               (* Тиск масла % *)
    PHY_SteamPressure   : INT;               (* Тиск пари бар *)

    (* Детектори фронтів для імпульсних входів *)
    FF_StartOld         : BOOL := FALSE;
    FF_StopOld          : BOOL := FALSE;
    FF_ResetOld         : BOOL := FALSE;
    FF_GasOld           : BOOL := FALSE;
    FF_VacuumOld        : BOOL := FALSE;
    FF_AlarmOld         : BOOL := FALSE;

    (* Лічильники та статистика *)
    CNT_Starts          : INT := 0;
    CNT_Stops           : INT := 0;
    CNT_Alarms          : INT := 0;
    CNT_GasFailures     : INT := 0;
    CNT_VacuumFailures  : INT := 0;
    CNT_RunTime         : INT := 0;          (* Час роботи в секундах *)
    TMR_RunTimer        : TON;               (* Таймер роботи *)

    (* Таймери та затримки *)
    TMR_StartDelay      : TON;               (* Затримка старту 3с *)
    TMR_AlarmDelay      : TON;               (* Затримка аварії 2с *)
    TMR_ResetDelay      : TON;               (* Затримка скидання 1с *)
END_VAR

(* ============================================
   ОСНОВНА ЛОГІКА ПРОГРАМИ
   ============================================ *)

(* --- БЛОК 1: ПЕРЕТВОРЕННЯ АЦП У ФІЗИЧНІ ВЕЛИЧИНИ --- *)
PHY_Voltage := AI_BoilerVoltage * VOLTAGE_MAX / ADC_MAX;
PHY_BoilerTemp := AI_BoilerTemp * TEMP_MAX / ADC_MAX;
PHY_WaterTemp := AI_WaterTemp * TEMP_MAX / ADC_MAX;
PHY_Temp1 := AI_TempSensor1 * TEMP_MAX / ADC_MAX;
PHY_Temp2 := AI_TempSensor2 * TEMP_MAX / ADC_MAX;
PHY_OilPressure := AI_OilPressure * 100 / ADC_MAX;
PHY_SteamPressure := AI_SteamPressure * 10 / ADC_MAX;

(* --- БЛОК 2: ЧИТАННЯ ДИСКРЕТНИХ ДАТЧИКІВ --- *)
SNS_GasPresent := DI_GasSensor;          (* 1 = газ є, 0 = немає *)
SNS_VacuumPresent := DI_VacuumSensor;     (* 1 = вакуум є, 0 = немає *)
SNS_OilPressureOK := DI_OilPressureOK;    (* 1 = норма, 0 = аварія *)
SNS_SteamPressureOK := DI_SteamPressureOK; (* 1 = норма, 0 = аварія *)
SYS_ManualMode := DI_ManualMode;

(* --- БЛОК 3: АВАРІЯ ВИСОКОЇ НАПРУГИ (≥400В) --- *)
IF PHY_Voltage >= VOLTAGE_TRIP THEN
    ALM_VoltageHigh := TRUE;
ELSE
    IF PHY_Voltage < VOLTAGE_RESET THEN
        ALM_VoltageHigh := FALSE;
    END_IF;
END_IF;

(* --- БЛОК 4: АВАРІЯ ВИСОКОЇ ТЕМПЕРАТУРИ (≥80°C) --- *)
IF PHY_BoilerTemp >= TEMP_TRIP THEN
    ALM_TempHigh := TRUE;
ELSE
    IF PHY_BoilerTemp < TEMP_RESET THEN
        ALM_TempHigh := FALSE;
    END_IF;
END_IF;

(* --- БЛОК 5: АВАРІЇ ПО ДАТЧИКАХ --- *)
ALM_NoGas := NOT SNS_GasPresent;           (* Немає газу = аварія *)
ALM_NoVacuum := NOT SNS_VacuumPresent;     (* Немає вакууму = аварія *)
ALM_OilPressureLow := NOT SNS_OilPressureOK; (* Низький тиск масла = аварія *)
ALM_SteamPressureBad := NOT SNS_SteamPressureOK; (* Неправильний тиск пари = аварія *)
ALM_Emergency := DI_EmergencyStop;         (* Зовнішній аварійний стоп *)

(* --- БЛОК 6: ЗАГАЛЬНА АВАРІЯ --- *)
ALM_AnyAlarm := ALM_VoltageHigh
              OR ALM_TempHigh
              OR ALM_NoGas
              OR ALM_NoVacuum
              OR ALM_OilPressureLow
              OR ALM_SteamPressureBad
              OR ALM_Emergency;

(* --- БЛОК 7: ЛОГІКА СТАРТ/СТОП --- *)

(* Детектор фронту команди старт *)
IF CMD_SystemStart AND NOT FF_StartOld THEN
    IF NOT SYS_Running AND NOT ALM_AnyAlarm THEN
        SYS_Enabled := TRUE;
        TMR_StartDelay(IN := TRUE, PT := T#3S); (* Затримка старту 3 секунди *)
    END_IF;
END_IF;
FF_StartOld := CMD_SystemStart;

(* Детектор фронту команди стоп *)
IF CMD_SystemStop AND NOT FF_StopOld THEN
    SYS_Enabled := FALSE;
    SYS_Running := FALSE;
END_IF;
FF_StopOld := CMD_SystemStop;

(* Автоматичний стоп при будь-якій аварії - НЕГАЙНО! *)
IF ALM_AnyAlarm THEN
    SYS_Enabled := FALSE;
    SYS_Running := FALSE;
END_IF;

(* Запуск після затримки *)
IF TMR_StartDelay.Q THEN
    SYS_Running := TRUE;
    TMR_StartDelay(IN := FALSE);
    CNT_Starts := CNT_Starts + 1;
END_IF;

(* --- БЛОК 8: ГОТОВНІСТЬ СИСТЕМИ --- *)
SYS_Ready := NOT ALM_VoltageHigh
           AND NOT ALM_TempHigh
           AND SNS_GasPresent
           AND SNS_VacuumPresent
           AND SNS_OilPressureOK
           AND SNS_SteamPressureOK
           AND NOT ALM_Emergency
           AND SYS_Running;

(* --- БЛОК 9: КЕРУВАННЯ КЛАПАНОМ ГАЗУ --- *)
(* ГОЛОВНЕ ПРАВИЛО: Газ відкритий тільки якщо ВСІ умови виконані *)
IF SYS_Ready THEN
    DO_GasValve := TRUE;    (* Відкрити клапан газу *)
ELSE
    DO_GasValve := FALSE;   (* ЗАКРИТИ клапан газу *)
END_IF;

(* ДОДАТКОВИЙ ЗАХИСТ: Якщо немає вакууму - ОБОВ'ЯЗКОВО закрити газ *)
IF NOT SNS_VacuumPresent THEN
    DO_GasValve := FALSE;
END_IF;

(* --- БЛОК 10: КЕРУВАННЯ РОЗЕТКАМИ --- *)
(* Розетки працюють тільки якщо немає аварій *)
DO_Socket1 := CMD_Socket1_On AND NOT ALM_AnyAlarm;
DO_Socket2 := CMD_Socket2_On AND NOT ALM_AnyAlarm;

(* --- БЛОК 11: КЕРУВАННЯ НАСОСАМИ --- *)
(* Насос води: працює якщо система готова і є температура води *)
DO_WaterPump := SYS_Ready AND PHY_WaterTemp > 20;

(* Насос масла: працює якщо система готова і тиск в нормі *)
DO_OilPump := SYS_Ready AND SNS_OilPressureOK;

(* Вентиляція: працює коли система працює *)
DO_FanVent := SYS_Running;

(* --- БЛОК 12: СИГНАЛІЗАЦІЯ ТА ІНДИКАЦІЯ --- *)
DO_AlarmLight := ALM_AnyAlarm;              (* Аварійна лампа *)
DO_PermitRun := SYS_Ready;                 (* Дозвіл роботи *)

(* Вивід стану для HMI *)
ST_SystemRunning := INT#1 IF SYS_Running ELSE INT#0;
ST_GasAvailable := INT#1 IF SNS_GasPresent ELSE INT#0;
ST_VacuumOK := INT#1 IF SNS_VacuumPresent ELSE INT#0;

(* Коди аварій для HMI *)
IF ALM_VoltageHigh THEN ST_AlarmCode := 1;
ELSIF ALM_TempHigh THEN ST_AlarmCode := 2;
ELSIF ALM_NoGas THEN ST_AlarmCode := 3;
ELSIF ALM_NoVacuum THEN ST_AlarmCode := 4;
ELSIF ALM_OilPressureLow THEN ST_AlarmCode := 5;
ELSIF ALM_SteamPressureBad THEN ST_AlarmCode := 6;
ELSIF ALM_Emergency THEN ST_AlarmCode := 7;
ELSE ST_AlarmCode := 0;
END_IF;

(* --- БЛОК 13: СТАТИСТИКА ТА ЛІЧИЛЬНИКИ --- *)

(* Лічильник аварій по передньому фронту *)
IF ALM_AnyAlarm AND NOT FF_AlarmOld THEN
    CNT_Alarms := CNT_Alarms + 1;
END_IF;
FF_AlarmOld := ALM_AnyAlarm;

(* Лічильник відмов газу *)
IF NOT SNS_GasPresent AND FF_GasOld THEN
    CNT_GasFailures := CNT_GasFailures + 1;
END_IF;
FF_GasOld := SNS_GasPresent;

(* Лічильник відмов вакууму *)
IF NOT SNS_VacuumPresent AND FF_VacuumOld THEN
    CNT_VacuumFailures := CNT_VacuumFailures + 1;
END_IF;
FF_VacuumOld := SNS_VacuumPresent;

(* Лічильник зупинок *)
IF (CMD_SystemStop AND NOT FF_StopOld) OR (ALM_AnyAlarm AND NOT FF_AlarmOld) THEN
    IF SYS_Running THEN
        CNT_Stops := CNT_Stops + 1;
    END_IF;
END_IF;

(* Таймер роботи системи *)
TMR_RunTimer(IN := SYS_Running, PT := T#1S);
IF TMR_RunTimer.Q THEN
    CNT_RunTime := CNT_RunTime + 1;
    TMR_RunTimer(IN := FALSE);
    TMR_RunTimer(IN := TRUE);
END_IF;

(* --- БЛОК 14: СКИДАННЯ АВАРІЙ --- *)
IF CMD_ResetAlarms AND NOT FF_ResetOld THEN
    TMR_ResetDelay(IN := TRUE, PT := T#1S);
END_IF;
FF_ResetOld := CMD_ResetAlarms;

IF TMR_ResetDelay.Q THEN
    (* Скидаємо тільки ті аварії, які можна скинути вручну *)
    IF NOT ALM_VoltageHigh AND NOT ALM_TempHigh AND NOT ALM_Emergency THEN
        ALM_NoGas := FALSE;
        ALM_NoVacuum := FALSE;
        ALM_OilPressureLow := FALSE;
        ALM_SteamPressureBad := FALSE;
    END_IF;
    TMR_ResetDelay(IN := FALSE);
END_IF;

(* ============================================
   ЕКСПОРТ ДАНИХ ДЛЯ HMI (REGISTRI)
   ============================================ *)
(* Аналогові дані для відображення *)
(*
MW0  = PHY_Voltage        (* Напруга бойлера В *)
MW1  = PHY_BoilerTemp     (* Температура бойлера °C *)
MW2  = PHY_WaterTemp      (* Температура води °C *)
MW3  = PHY_Temp1          (* Температура датчик 1 °C *)
MW4  = PHY_Temp2          (* Температура датчик 2 °C *)
MW5  = PHY_OilPressure    (* Тиск масла % *)
MW6  = PHY_SteamPressure  (* Тиск пари бар *)

MW10 = CNT_Starts         (* Кількість запусків *)
MW11 = CNT_Stops          (* Кількість зупинок *)
MW12 = CNT_Alarms         (* Кількість аварій *)
MW13 = CNT_GasFailures    (* Відмов газу *)
MW14 = CNT_VacuumFailures (* Відмов вакууму *)
MW15 = CNT_RunTime        (* Час роботи секунд *)

MX20 = SYS_Running         (* Система працює *)
MX21 = SYS_Ready          (* Система готова *)
MX22 = SNS_GasPresent     (* Газ присутній *)
MX23 = SNS_VacuumPresent  (* Вакуум присутній *)
MX24 = ALM_VoltageHigh    (* Аварія напруги *)
MX25 = ALM_TempHigh       (* Аварія температури *)
MX26 = ALM_NoGas          (* Аварія газу *)
MX27 = ALM_NoVacuum       (* Аварія вакууму *)
MX28 = ALM_OilPressureLow (* Аварія тиску масла *)
MX29 = ALM_SteamPressureBad(* Аварія тиску пари *)
MX30 = ALM_Emergency      (* Аварійний стоп *)
MX31 = ALM_AnyAlarm       (* Будь-яка аварія *)
*)

END_PROGRAM

(* ---- FATEK_BoilerControl_Safe.ST ---- *)
(* ============================================
   ДОДАТКОВИЙ ЗАХИСТ ДЛЯ FATEK FBs-10MAR
   Розширена версія з додатковими перевірками
   ============================================ *)

PROGRAM BoilerControlSafe

(* --- ДОДАТКОВІ КОНСТАНТИ БЕЗПЕКИ --- *)
VAR_CONSTANT
    (* Межі АЦП з запасом *)
    ADC_SAFE_MIN        : INT := 100;           (* Мінімальне значення АЦП *)
    ADC_SAFE_MAX        : INT := 3900;          (* Максимальне значення АЦП *)

    (* Діапазони перевірки датчиків *)
    VOLTAGE_MIN_CHECK   : INT := 50;            (* Мінімальна напруга 50В *)
    VOLTAGE_MAX_CHECK   : INT := 480;           (* Максимальна напруга 480В *)
    TEMP_MIN_CHECK      : INT := -20;           (* Мінімальна температура -20°C *)
    TEMP_MAX_CHECK      : INT := 120;           (* Максимальна температура 120°C *)

    (* Часові затримки безпеки *)
    STARTUP_DELAY       : TIME := T#5S;         (* Затримка старту 5 секунд *)
    GAS_VALVE_DELAY     : TIME := T#2S;         (* Затримка відкриття газу 2с *)
    EMERGENCY_SHUTDOWN  : TIME := T#0.5S;       (* Аварійне відключення 0.5с *)

    (* Кількість циклів для стабілізації *)
    STABILIZATION_CYCLES: INT := 10;            (* 10 циклів для стабілізації *)
END_VAR

(* --- ДОДАТКОВІ МАРКЕРИ БЕЗПЕКИ --- *)
VAR
    (* Перевірка датчиків *)
    SNS_VoltageOK       : BOOL := TRUE;         (* Напруга в межах норми *)
    SNS_TemperatureOK   : BOOL := TRUE;         (* Температура в межах норми *)
    SNS_ADC_OK          : BOOL := TRUE;         (* АЦП працює нормально *)
    SNS_CommunicationOK : BOOL := TRUE;         (* Зв'язок з датчиками є *)

    (* Стани безпеки *)
    SAF_SystemStable    : BOOL := FALSE;        (* Система стабілізована *)
    SAF_StartupMode      : BOOL := TRUE;         (* Режим старту *)
    SAF_EmergencyMode   : BOOL := FALSE;        (* Аварійний режим *)
    SAF_ManualOverride  : BOOL := FALSE;        (* Ручне перевизначення *)

    (* Лічильники безпеки *)
    SAF_CycleCounter    : INT := 0;             (* Лічильник циклів *)
    SAF_ErrorCounter    : INT := 0;             (* Лічильник помилок *)
    SAF_LastErrorTime   : TIME := T#0S;         (* Час останньої помилки *)

    (* Детектори помилок *)
    ERR_ADC_Failure     : BOOL := FALSE;        (* Відмова АЦП *)
    ERR_SensorRange     : BOOL := FALSE;        (* Датчик поза діапазоном *)
    ERR_CommTimeout     : BOOL := FALSE;        (* Тайм-аут зв'язку *)
    ERR_PowerSupply     : BOOL := FALSE;        (* Проблема живлення *)

    (* Таймери безпеки *)
    TMR_SafetyStartup   : TON;                  (* Таймер безпечного старту *)
    TMR_GasValveSafety  : TON;                  (* Таймер безпеки газового клапана *)
    TMR_EmergencyDelay  : TON;                  (* Таймер аварійної затримки *)
    TMR_Watchdog        : TON;                  (* Ватчдог системи *)

    (* Буфери для фільтрації *)
    FILTER_Voltage      : ARRAY[0..4] OF INT;   (* Фільтр напруги *)
    FILTER_Temperature  : ARRAY[0..4] OF INT;   (* Фільтр температури *)
    FILTER_Index        : INT := 0;             (* Індекс фільтра *)
END_VAR

(* ============================================
   БЛОК БЕЗПЕКИ: ПЕРЕВІРКА АЦП ВХОДІВ
   ============================================ *)

(* Перевірка АЦП на вихід за межі *)
IF (AI_BoilerVoltage < ADC_SAFE_MIN OR AI_BoilerVoltage > ADC_SAFE_MAX) OR
   (AI_BoilerTemp < ADC_SAFE_MIN OR AI_BoilerTemp > ADC_SAFE_MAX) OR
   (AI_WaterTemp < ADC_SAFE_MIN OR AI_WaterTemp > ADC_SAFE_MAX) THEN
    ERR_ADC_Failure := TRUE;
    SAF_ErrorCounter := SAF_ErrorCounter + 1;
ELSE
    ERR_ADC_Failure := FALSE;
END_IF;

(* Перевірка фізичних величин на адекватність *)
IF (PHY_Voltage < VOLTAGE_MIN_CHECK OR PHY_Voltage > VOLTAGE_MAX_CHECK) OR
   (PHY_BoilerTemp < TEMP_MIN_CHECK OR PHY_BoilerTemp > TEMP_MAX_CHECK) THEN
    ERR_SensorRange := TRUE;
    SAF_ErrorCounter := SAF_ErrorCounter + 1;
ELSE
    ERR_SensorRange := FALSE;
END_IF;

(* ============================================
   БЛОК БЕЗПЕКИ: ФІЛЬТРАЦІЯ СИГНАЛІВ
   ============================================ *)

(* Кільцевий буфер для фільтрації напруги *)
FILTER_Voltage[FILTER_Index] := AI_BoilerVoltage;
FILTER_Temperature[FILTER_Index] := AI_BoilerTemp;

(* Обчислення середнього значення *)
VAR
    i : INT;
    sum_voltage : INT := 0;
    sum_temp : INT := 0;
END_VAR

FOR i := 0 TO 4 DO
    sum_voltage := sum_voltage + FILTER_Voltage[i];
    sum_temp := sum_temp + FILTER_Temperature[i];
END_FOR;

(* Використовуємо відфільтровані значення *)
PHY_Voltage := (sum_voltage / 5) * VOLTAGE_MAX / ADC_MAX;
PHY_BoilerTemp := (sum_temp / 5) * TEMP_MAX / ADC_MAX;

(* Оновлення індексу фільтра *)
FILTER_Index := (FILTER_Index + 1) MOD 5;

(* ============================================
   БЛОК БЕЗПЕКИ: СТАБІЛІЗАЦІЯ СИСТЕМИ
   ============================================ *)

(* Лічильник циклів для стабілізації *)
IF SAF_CycleCounter < STABILIZATION_CYCLES THEN
    SAF_CycleCounter := SAF_CycleCounter + 1;
    SAF_SystemStable := FALSE;
    SAF_StartupMode := TRUE;
ELSE
    SAF_SystemStable := TRUE;
    SAF_StartupMode := FALSE;
END_IF;

(* Таймер безпечного старту *)
TMR_SafetyStartup(IN := SAF_StartupMode, PT := STARTUP_DELAY);

(* ============================================
   БЛОК БЕЗПЕКИ: УМОВИ РОБОТИ
   ============================================ *)

(* Загальні умови безпеки *)
SNS_VoltageOK := NOT ERR_ADC_Failure AND NOT ERR_SensorRange;
SNS_TemperatureOK := NOT ERR_SensorRange;
SNS_ADC_OK := NOT ERR_ADC_Failure;
SNS_CommunicationOK := TRUE; (* Для майбутнього розширення *)

(* ============================================
   БЛОК БЕЗПЕКИ: МОДИФІКОВАНА ЛОГІКА УПРАВЛІННЯ
   ============================================ *)

(* Посилені умови готовності системи *)
SYS_Ready := SAF_SystemStable                    (* Система стабільна *)
           AND SNS_VoltageOK                      (* Напруга норма *)
           AND SNS_TemperatureOK                  (* Температура норма *)
           AND SNS_ADC_OK                         (* АЦП працює *)
           AND NOT ERR_ADC_Failure                (* Немає помилок АЦП *)
           AND NOT ERR_SensorRange                (* Датчики в діапазоні *)
           AND NOT SAF_EmergencyMode              (* Не аварійний режим *)
           AND SNS_GasPresent                      (* Газ є *)
           AND SNS_VacuumPresent                   (* Вакуум є *)
           AND SNS_OilPressureOK                   (* Тиск масла норма *)
           AND SNS_SteamPressureOK                 (* Тиск пари норма *)
           AND NOT ALM_Emergency                   (* Немає зовнішньої аварії *)
           AND SYS_Running                         (* Система запущена *)
           AND SAF_ErrorCounter < 10;              (* Забагато помилок? *)

(* ============================================
   БЛОК БЕЗПЕКИ: КЕРУВАННЯ ГАЗОВИМ КЛАПАНОМ
   ============================================ *)

(* Додатковий таймер безпеки для газового клапана *)
IF SYS_Ready THEN
    TMR_GasValveSafety(IN := TRUE, PT := GAS_VALVE_DELAY);
ELSE
    TMR_GasValveSafety(IN := FALSE);
END_IF;

(* Відкриття газу тільки після всіх перевірок + затримка *)
DO_GasValve := SYS_Ready AND TMR_GasValveSafety.Q AND NOT SAF_StartupMode;

(* ПРИОРИТЕТНИЙ ЗАХИСТ: Вакуум важливіший за все! *)
IF NOT SNS_VacuumPresent THEN
    DO_GasValve := FALSE;
    SAF_EmergencyMode := TRUE;
END_IF;

(* ============================================
   БЛОК БЕЗПЕКИ: АВАРІЙНІ ВИХОДИ
   ============================================ *)

(* Аварійне відключення при критичних помилках *)
IF ERR_ADC_Failure OR ERR_SensorRange OR SAF_ErrorCounter >= 10 THEN
    SAF_EmergencyMode := TRUE;
    TMR_EmergencyDelay(IN := TRUE, PT := EMERGENCY_SHUTDOWN);
END_IF;

(* Примусове відключення всього при аварії *)
IF SAF_EmergencyMode OR TMR_EmergencyDelay.Q THEN
    DO_GasValve := FALSE;
    DO_Socket1 := FALSE;
    DO_Socket2 := FALSE;
    DO_WaterPump := FALSE;
    DO_OilPump := FALSE;
    DO_FanVent := FALSE;
    SYS_Running := FALSE;
END_IF;

(* ============================================
   БЛОК БЕЗПЕКИ: WATCHDOG ТА ДІАГНОСТИКА
   ============================================ *)

(* Watchdog таймер - має перезавантажуватись кожен цикл *)
TMR_Watchdog(IN := TRUE, PT := T#1S);

(* Якщо watchdog не спрацьовує - є проблема з циклом сканування *)
IF NOT TMR_Watchdog.Q THEN
    ERR_CommTimeout := TRUE;
    SAF_ErrorCounter := SAF_ErrorCounter + 1;
END_IF;

(* Скидання watchdog на кожному циклі *)
TMR_Watchdog(IN := FALSE);
TMR_Watchdog(IN := TRUE);

(* ============================================
   БЛОК БЕЗПЕКИ: ІНДИКАЦІЯ ПОМИЛОК
   ============================================ *)

(* Розширена індикація кодів помилок *)
IF ERR_ADC_Failure THEN ST_AlarmCode := 10;
ELSIF ERR_SensorRange THEN ST_AlarmCode := 11;
ELSIF ERR_CommTimeout THEN ST_AlarmCode := 12;
ELSIF ERR_PowerSupply THEN ST_AlarmCode := 13;
ELSIF SAF_EmergencyMode THEN ST_AlarmCode := 99;
ELSE
    (* Оригінальні коди аварій *)
    IF ALM_VoltageHigh THEN ST_AlarmCode := 1;
    ELSIF ALM_TempHigh THEN ST_AlarmCode := 2;
    ELSIF ALM_NoGas THEN ST_AlarmCode := 3;
    ELSIF ALM_NoVacuum THEN ST_AlarmCode := 4;
    ELSIF ALM_OilPressureLow THEN ST_AlarmCode := 5;
    ELSIF ALM_SteamPressureBad THEN ST_AlarmCode := 6;
    ELSIF ALM_Emergency THEN ST_AlarmCode := 7;
    ELSE ST_AlarmCode := 0;
    END_IF;
END_IF;

(* ============================================
   БЛОК БЕЗПЕКИ: ЛОГІКУВАННЯ ПОМИЛОК
   ============================================ *)

(* Реєстрація часу помилки *)
IF ERR_ADC_Failure OR ERR_SensorRange OR ERR_CommTimeout THEN
    SAF_LastErrorTime := CURRENT_TIME;
END_IF;

(* Автоматичне скидання помилок після 5 хвилин *)
IF (CURRENT_TIME - SAF_LastErrorTime) > T#5M THEN
    ERR_ADC_Failure := FALSE;
    ERR_SensorRange := FALSE;
    ERR_CommTimeout := FALSE;
    SAF_EmergencyMode := FALSE;
    SAF_ErrorCounter := 0;
END_IF;

END_PROGRAM

(* ---- WinProladder.ST ---- *)
(* ============================================
   КЕРУВАННЯ БОЙЛЕРОМ / ГАЗОВИМ ОБЛАДНАННЯМ
   Fatek FBs-MA — Structured Text (ST)
   ============================================ *)

(* --- КОНСТАНТИ --- *)
VAR CONSTANT
    NAPRUGA_AVARIA      : INT := 3276;  (* 400В → АЦП: 4095*400/500=3276 *)
    TEMP_BOILER_AVARIA  : INT := 2184;  (* 80°C → АЦП: 4095*80/150=2184 *)
END_VAR

(* --- ЗМІННІ ВХОДІВ (Inputs) --- *)
VAR
    (* Аналогові входи 0..4095 *)
    AI_NAPRUGA      AT %IW0 : INT;   (* Напруга бойлера через перетворювач *)
    AI_TEMP_BOILER  AT %IW1 : INT;   (* Температура бойлера PT100/4-20mA *)
    AI_TEMP_VODA    AT %IW2 : INT;   (* Температура води *)
    AI_TEMP_2       AT %IW3 : INT;   (* Додатковий датчик температури *)
    AI_TISK_MASLA   AT %IW4 : INT;   (* Тиск масла (аналог) *)

    (* Дискретні входи *)
    X_GAZ           AT %IX0.0 : BOOL; (* Датчик газу: TRUE=є газ (замкнутий) *)
    X_VAKUUM        AT %IX0.1 : BOOL; (* Датчик вакууму: TRUE=є вакуум *)
    X_TISK_MASLA_DI AT %IX0.2 : BOOL; (* Тиск масла дискретний: TRUE=норма *)
    X_AVARIA_EXT    AT %IX0.3 : BOOL; (* Зовнішній аварійний стоп *)

    (* Команди з HMI / оператора *)
    CMD_ROZET_1     AT %MX10.0 : BOOL; (* Команда вкл. розетки 1 *)
    CMD_ROZET_2     AT %MX10.1 : BOOL; (* Команда вкл. розетки 2 *)
    CMD_START       AT %MX10.2 : BOOL; (* Старт системи *)
    CMD_STOP        AT %MX10.3 : BOOL; (* Стоп системи *)
END_VAR

(* --- ЗМІННІ ВИХОДІВ (Outputs) --- *)
VAR
    Y_KLAPAN_GAZ    AT %QX0.0 : BOOL; (* Клапан газу: TRUE=відкрито *)
    Y_ROZET_1       AT %QX0.1 : BOOL; (* Розетка 1 *)
    Y_ROZET_2       AT %QX0.2 : BOOL; (* Розетка 2 *)
    Y_AVARIA_SIGNAL AT %QX0.3 : BOOL; (* Аварійна сигналізація *)
    Y_DOZV_ROBOTY   AT %QX0.4 : BOOL; (* Загальний дозвіл роботи *)
END_VAR

(* --- ВНУТРІШНІ МАРКЕРИ --- *)
VAR
    M_AVARIA_NAPRUGA    : BOOL; (* Аварія: напруга >= 400В *)
    M_AVARIA_TEMP       : BOOL; (* Аварія: температура >= 80°C *)
    M_GAZ_IE            : BOOL; (* Газ є = 1, немає = 0 *)
    M_VAKUUM_IE         : BOOL; (* Вакуум є = 1, немає = 0 *)
    M_TISK_NORMA        : BOOL; (* Тиск масла в нормі *)
    M_AVARIA_VAKUUM     : BOOL; (* Аварія: пропав вакуум *)
    M_SYSTEM_READY      : BOOL; (* Система готова до роботи *)
    M_ZAGALNA_AVARIA    : BOOL; (* Будь-яка аварія *)
    M_SYSTEM_ON         : BOOL; (* Система запущена *)

    (* Температури в градусах для відображення *)
    TEMP_BOILER_GRAD    : INT;  (* Температура бойлера °C *)
    TEMP_VODA_GRAD      : INT;  (* Температура води °C *)
    TEMP_2_GRAD         : INT;  (* Температура доп. датчик °C *)
    NAPRUGA_VOLT        : INT;  (* Напруга в Вольтах *)
END_VAR

(* ============================================
   БЛОК 1: СТАРТ / СТОП СИСТЕМИ
   ============================================ *)
IF CMD_START AND NOT CMD_STOP AND NOT M_ZAGALNA_AVARIA THEN
    M_SYSTEM_ON := TRUE;
END_IF;

IF CMD_STOP OR M_ZAGALNA_AVARIA THEN
    M_SYSTEM_ON := FALSE;
END_IF;

(* ============================================
   БЛОК 2: ПЕРЕРАХУНОК АЦП → РЕАЛЬНІ ОДИНИЦІ
   Формула: РЕАЛ = АЦП * MAX_ЗНАЧЕННЯ / 4095
   ============================================ *)

(* Напруга: 0-4095 = 0-500В *)
NAPRUGA_VOLT    := AI_NAPRUGA    * 500 / 4095;

(* Температури: 0-4095 = 0-150°C *)
TEMP_BOILER_GRAD := AI_TEMP_BOILER * 150 / 4095;
TEMP_VODA_GRAD   := AI_TEMP_VODA   * 150 / 4095;
TEMP_2_GRAD      := AI_TEMP_2      * 150 / 4095;

(* ============================================
   БЛОК 3: АВАРІЯ ПО НАПРУЗІ БОЙЛЕРА
   Якщо напруга >= 400В → АВАРІЯ → ЗУПИНКА
   ============================================ *)
IF NAPRUGA_VOLT >= 400 THEN
    M_AVARIA_NAPRUGA := TRUE;
ELSE
    (* Гістерезис: скидати тільки якщо впала нижче 380В *)
    IF NAPRUGA_VOLT < 380 THEN
        M_AVARIA_NAPRUGA := FALSE;
    END_IF;
END_IF;

(* ============================================
   БЛОК 4: АВАРІЯ ПО ТЕМПЕРАТУРІ БОЙЛЕРА
   Якщо температура >= 80°C → АВАРІЯ → ЗУПИНКА
   ============================================ *)
IF TEMP_BOILER_GRAD >= 80 THEN
    M_AVARIA_TEMP := TRUE;
ELSE
    (* Гістерезис: скидати тільки якщо охолонув нижче 75°C *)
    IF TEMP_BOILER_GRAD < 75 THEN
        M_AVARIA_TEMP := FALSE;
    END_IF;
END_IF;

(* ============================================
   БЛОК 5: ДАТЧИК ГАЗУ
   X_GAZ = TRUE (замкнутий) → газ є (M_GAZ_IE = 1)
   X_GAZ = FALSE (розімкнутий) → газу немає (M_GAZ_IE = 0)
   ============================================ *)
M_GAZ_IE := X_GAZ;

(* ============================================
   БЛОК 6: ДАТЧИК ВАКУУМУ
   X_VAKUUM = TRUE (замкнутий) → вакуум є
   X_VAKUUM = FALSE (розімкнутий) → вакууму немає → ЗУПИНКА
   ============================================ *)
M_VAKUUM_IE := X_VAKUUM;

IF NOT M_VAKUUM_IE THEN
    M_AVARIA_VAKUUM := TRUE;  (* Пропав вакуум — аварія *)
ELSE
    M_AVARIA_VAKUUM := FALSE; (* Вакуум є — норма *)
END_IF;

(* ============================================
   БЛОК 7: ТИСК МАСЛА
   X_TISK_MASLA_DI = TRUE → тиск норма
   ============================================ *)
M_TISK_NORMA := X_TISK_MASLA_DI;

(* ============================================
   БЛОК 8: ЗАГАЛЬНА АВАРІЯ
   Будь-яка з умов → загальна аварія
   ============================================ *)
M_ZAGALNA_AVARIA := M_AVARIA_NAPRUGA
                 OR M_AVARIA_TEMP
                 OR M_AVARIA_VAKUUM
                 OR NOT M_TISK_NORMA
                 OR X_AVARIA_EXT;

(* ============================================
   БЛОК 9: ГОТОВНІСТЬ СИСТЕМИ ДО РОБОТИ
   Всі умови мають бути виконані
   ============================================ *)
M_SYSTEM_READY := NOT M_AVARIA_NAPRUGA   (* Напруга норма *)
              AND NOT M_AVARIA_TEMP       (* Температура норма *)
              AND M_GAZ_IE                (* Газ є *)
              AND M_VAKUUM_IE             (* Вакуум є *)
              AND M_TISK_NORMA            (* Тиск масла норма *)
              AND NOT X_AVARIA_EXT        (* Немає зовнішньої аварії *)
              AND M_SYSTEM_ON;            (* Система запущена *)

(* ============================================
   БЛОК 10: КЕРУВАННЯ КЛАПАНОМ ГАЗУ (Y0)
   Відкрити тільки якщо ВСІ умови виконані:
   - є газ
   - є вакуум  ← КРИТИЧНО: без вакууму ЗАЧИНИТИ!
   - немає аварії напруги
   - немає аварії температури
   - тиск масла норма
   - система запущена
   ============================================ *)
IF M_SYSTEM_READY THEN
    Y_KLAPAN_GAZ := TRUE;   (* Відкрити клапан газу *)
ELSE
    Y_KLAPAN_GAZ := FALSE;  (* ЗАЧИНИТИ клапан газу *)
END_IF;

(* Додаткова гарантія: якщо немає вакууму — ОБОВ'ЯЗКОВО закрити газ *)
IF NOT M_VAKUUM_IE THEN
    Y_KLAPAN_GAZ := FALSE;
END_IF;

(* ============================================
   БЛОК 11: КЕРУВАННЯ РОЗЕТКАМИ
   Вмикаються командою з контролера/HMI
   але тільки якщо немає загальної аварії
   ============================================ *)
IF CMD_ROZET_1 AND NOT M_ZAGALNA_AVARIA THEN
    Y_ROZET_1 := TRUE;
ELSE
    Y_ROZET_1 := FALSE;
END_IF;

IF CMD_ROZET_2 AND NOT M_ZAGALNA_AVARIA THEN
    Y_ROZET_2 := TRUE;
ELSE
    Y_ROZET_2 := FALSE;
END_IF;

(* ============================================
   БЛОК 12: АВАРІЙНА СИГНАЛІЗАЦІЯ
   ============================================ *)
Y_AVARIA_SIGNAL := M_ZAGALNA_AVARIA;

(* ============================================
   БЛОК 13: ЗАГАЛЬНИЙ ДОЗВІЛ РОБОТИ
   ============================================ *)
Y_DOZV_ROBOTY := M_SYSTEM_READY;
```

---

## 📋 Схема підключення входів/виходів
```
ВХОДИ (X / AI):
─────────────────────────────────────────────────────
 AI0  ← Перетворювач напруги (400В AC → 0-10V DC)
 AI1  ← Датчик температури бойлера (PT100 → 4-20mA модуль)
 AI2  ← Датчик температури води (PT100 → 4-20mA модуль)
 AI3  ← Датчик температури #2
 AI4  ← Датчик тиску масла (4-20mA)
 X0   ← Датчик ГАЗУ (кінцевий вимикач: замкн.=є газ)
 X1   ← Датчик ВАКУУМУ (кінцевий вимикач: замкн.=є вакуум)
 X2   ← Датчик ТИСКУ МАСЛА дискретний (замкн.=норма)
 X3   ← Кнопка аварійного СТОП

ВИХОДИ (Y):
─────────────────────────────────────────────────────
 Y0   → Соленоїдний КЛАПАН ГАЗУ (24VDC, через реле)
 Y1   → РОЗЕТКА 1 (через реле або SSR)
 Y2   → РОЗЕТКА 2 (через реле або SSR)
 Y3   → СИГНАЛІЗАЦІЯ аварії (лампа/сирена)
 Y4   → ДОЗВІЛ РОБОТИ (загальний контактор)

МАРКЕРИ для HMI дисплею:
─────────────────────────────────────────────────────
 MW0  = NAPRUGA_VOLT      (відображати в Вольтах)
 MW1  = TEMP_BOILER_GRAD  (відображати в °C)
 MW2  = TEMP_VODA_GRAD    (відображати в °C)
 MW3  = TEMP_2_GRAD       (відображати в °C)
 MX10.0 = CMD_ROZET_1     (кнопка вкл. розетки 1)
 MX10.1 = CMD_ROZET_2     (кнопка вкл. розетки 2)
 MX10.2 = CMD_START       (кнопка СТАРТ)
 MX10.3 = CMD_STOP        (кнопка СТОП)
